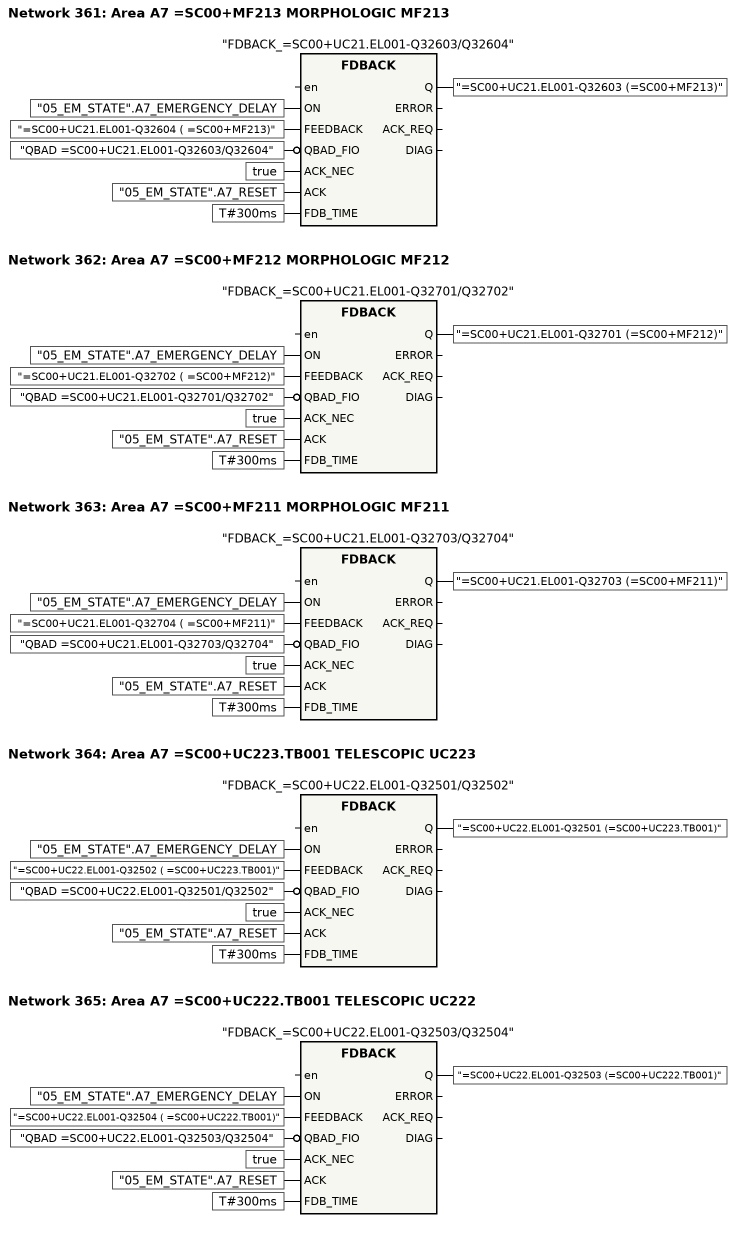
   "FDBACK_=SC00+UC21.EL001-Q32603/Q32604"(ON := "05_EM_STATE".A7_EMERGENCY_DELAY,   // FDBACK
                           FEEDBACK := "=SC00+UC21.EL001-Q32604 ( =SC00+MF213)",
                           QBAD_FIO := NOT "QBAD =SC00+UC21.EL001-Q32603/Q32604",
                           ACK_NEC := true,
                           ACK := "05_EM_STATE".A7_RESET,
                           FDB_TIME := T#300ms,
                           Q => "=SC00+UC21.EL001-Q32603 (=SC00+MF213)");
END_REGION

REGION Network 362: Area A7 =SC00+MF212 MORPHOLOGIC MF212
   "FDBACK_=SC00+UC21.EL001-Q32701/Q32702"(ON := "05_EM_STATE".A7_EMERGENCY_DELAY,   // FDBACK
                           FEEDBACK := "=SC00+UC21.EL001-Q32702 ( =SC00+MF212)",
                           QBAD_FIO := NOT "QBAD =SC00+UC21.EL001-Q32701/Q32702",
                           ACK_NEC := true,
                           ACK := "05_EM_STATE".A7_RESET,
                           FDB_TIME := T#300ms,
                           Q => "=SC00+UC21.EL001-Q32701 (=SC00+MF212)");
END_REGION

REGION Network 363: Area A7 =SC00+MF211 MORPHOLOGIC MF211
   "FDBACK_=SC00+UC21.EL001-Q32703/Q32704"(ON := "05_EM_STATE".A7_EMERGENCY_DELAY,   // FDBACK
                           FEEDBACK := "=SC00+UC21.EL001-Q32704 ( =SC00+MF211)",
                           QBAD_FIO := NOT "QBAD =SC00+UC21.EL001-Q32703/Q32704",
                           ACK_NEC := true,
                           ACK := "05_EM_STATE".A7_RESET,
                           FDB_TIME := T#300ms,
                           Q => "=SC00+UC21.EL001-Q32703 (=SC00+MF211)");
END_REGION

REGION Network 364: Area A7 =SC00+UC223.TB001 TELESCOPIC UC223
   "FDBACK_=SC00+UC22.EL001-Q32501/Q32502"(ON := "05_EM_STATE".A7_EMERGENCY_DELAY,   // FDBACK
                           FEEDBACK := "=SC00+UC22.EL001-Q32502 ( =SC00+UC223.TB001)",
                           QBAD_FIO := NOT "QBAD =SC00+UC22.EL001-Q32501/Q32502",
                           ACK_NEC := true,
                           ACK := "05_EM_STATE".A7_RESET,
                           FDB_TIME := T#300ms,
                           Q => "=SC00+UC22.EL001-Q32501 (=SC00+UC223.TB001)");
END_REGION

REGION Network 365: Area A7 =SC00+UC222.TB001 TELESCOPIC UC222
   "FDBACK_=SC00+UC22.EL001-Q32503/Q32504"(ON := "05_EM_STATE".A7_EMERGENCY_DELAY,   // FDBACK
                           FEEDBACK := "=SC00+UC22.EL001-Q32504 ( =SC00+UC222.TB001)",
                           QBAD_FIO := NOT "QBAD =SC00+UC22.EL001-Q32503/Q32504",
                           ACK_NEC := true,
                           ACK := "05_EM_STATE".A7_RESET,
                           FDB_TIME := T#300ms,
                           Q => "=SC00+UC22.EL001-Q32503 (=SC00+UC222.TB001)");
END_REGION

REGION Network 366: Area A7 =SC00+UC221.TB001 TELESCOPIC UC221
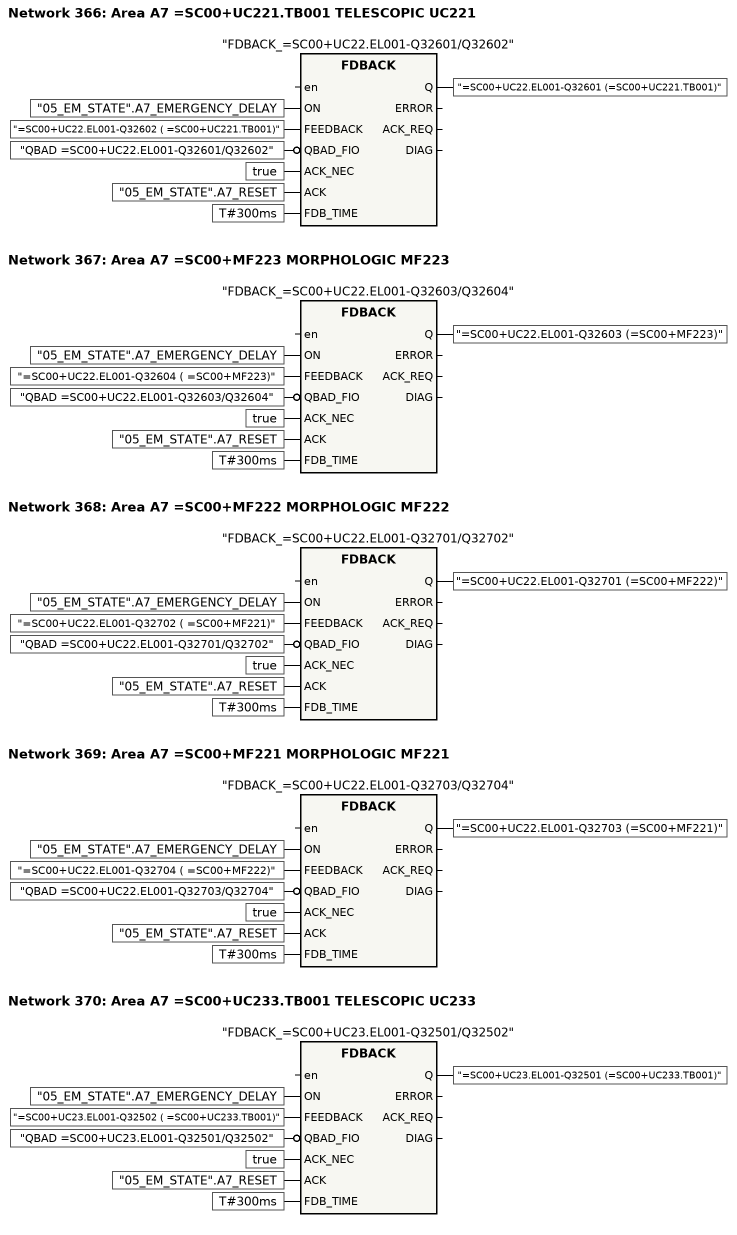
   "FDBACK_=SC00+UC22.EL001-Q32601/Q32602"(ON := "05_EM_STATE".A7_EMERGENCY_DELAY,   // FDBACK
                           FEEDBACK := "=SC00+UC22.EL001-Q32602 ( =SC00+UC221.TB001)",
                           QBAD_FIO := NOT "QBAD =SC00+UC22.EL001-Q32601/Q32602",
                           ACK_NEC := true,
                           ACK := "05_EM_STATE".A7_RESET,
                           FDB_TIME := T#300ms,
                           Q => "=SC00+UC22.EL001-Q32601 (=SC00+UC221.TB001)");
END_REGION

REGION Network 367: Area A7 =SC00+MF223 MORPHOLOGIC MF223
   "FDBACK_=SC00+UC22.EL001-Q32603/Q32604"(ON := "05_EM_STATE".A7_EMERGENCY_DELAY,   // FDBACK
                           FEEDBACK := "=SC00+UC22.EL001-Q32604 ( =SC00+MF223)",
                           QBAD_FIO := NOT "QBAD =SC00+UC22.EL001-Q32603/Q32604",
                           ACK_NEC := true,
                           ACK := "05_EM_STATE".A7_RESET,
                           FDB_TIME := T#300ms,
                           Q => "=SC00+UC22.EL001-Q32603 (=SC00+MF223)");
END_REGION

REGION Network 368: Area A7 =SC00+MF222 MORPHOLOGIC MF222
   "FDBACK_=SC00+UC22.EL001-Q32701/Q32702"(ON := "05_EM_STATE".A7_EMERGENCY_DELAY,   // FDBACK
                           FEEDBACK := "=SC00+UC22.EL001-Q32702 ( =SC00+MF221)",
                           QBAD_FIO := NOT "QBAD =SC00+UC22.EL001-Q32701/Q32702",
                           ACK_NEC := true,
                           ACK := "05_EM_STATE".A7_RESET,
                           FDB_TIME := T#300ms,
                           Q => "=SC00+UC22.EL001-Q32701 (=SC00+MF222)");
END_REGION

REGION Network 369: Area A7 =SC00+MF221 MORPHOLOGIC MF221
   "FDBACK_=SC00+UC22.EL001-Q32703/Q32704"(ON := "05_EM_STATE".A7_EMERGENCY_DELAY,   // FDBACK
                           FEEDBACK := "=SC00+UC22.EL001-Q32704 ( =SC00+MF222)",
                           QBAD_FIO := NOT "QBAD =SC00+UC22.EL001-Q32703/Q32704",
                           ACK_NEC := true,
                           ACK := "05_EM_STATE".A7_RESET,
                           FDB_TIME := T#300ms,
                           Q => "=SC00+UC22.EL001-Q32703 (=SC00+MF221)");
END_REGION

REGION Network 370: Area A7 =SC00+UC233.TB001 TELESCOPIC UC233
   "FDBACK_=SC00+UC23.EL001-Q32501/Q32502"(ON := "05_EM_STATE".A7_EMERGENCY_DELAY,   // FDBACK
                           FEEDBACK := "=SC00+UC23.EL001-Q32502 ( =SC00+UC233.TB001)",
                           QBAD_FIO := NOT "QBAD =SC00+UC23.EL001-Q32501/Q32502",
                           ACK_NEC := true,
                           ACK := "05_EM_STATE".A7_RESET,
                           FDB_TIME := T#300ms,
                           Q => "=SC00+UC23.EL001-Q32501 (=SC00+UC233.TB001)");
END_REGION

REGION Network 371: Area A7 =SC00+UC232.TB001 TELESCOPIC UC232
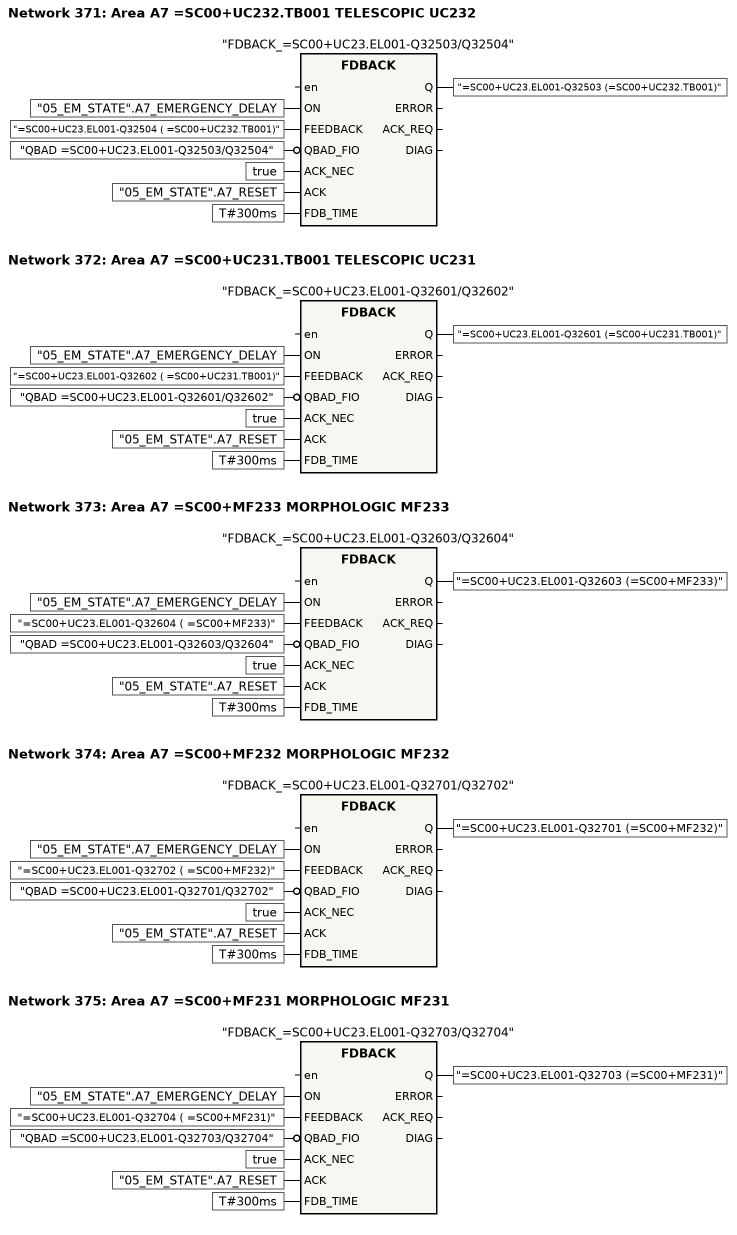
   "FDBACK_=SC00+UC23.EL001-Q32503/Q32504"(ON := "05_EM_STATE".A7_EMERGENCY_DELAY,   // FDBACK
                           FEEDBACK := "=SC00+UC23.EL001-Q32504 ( =SC00+UC232.TB001)",
                           QBAD_FIO := NOT "QBAD =SC00+UC23.EL001-Q32503/Q32504",
                           ACK_NEC := true,
                           ACK := "05_EM_STATE".A7_RESET,
                           FDB_TIME := T#300ms,
                           Q => "=SC00+UC23.EL001-Q32503 (=SC00+UC232.TB001)");
END_REGION

REGION Network 372: Area A7 =SC00+UC231.TB001 TELESCOPIC UC231
   "FDBACK_=SC00+UC23.EL001-Q32601/Q32602"(ON := "05_EM_STATE".A7_EMERGENCY_DELAY,   // FDBACK
                           FEEDBACK := "=SC00+UC23.EL001-Q32602 ( =SC00+UC231.TB001)",
                           QBAD_FIO := NOT "QBAD =SC00+UC23.EL001-Q32601/Q32602",
                           ACK_NEC := true,
                           ACK := "05_EM_STATE".A7_RESET,
                           FDB_TIME := T#300ms,
                           Q => "=SC00+UC23.EL001-Q32601 (=SC00+UC231.TB001)");
END_REGION

REGION Network 373: Area A7 =SC00+MF233 MORPHOLOGIC MF233
   "FDBACK_=SC00+UC23.EL001-Q32603/Q32604"(ON := "05_EM_STATE".A7_EMERGENCY_DELAY,   // FDBACK
                           FEEDBACK := "=SC00+UC23.EL001-Q32604 ( =SC00+MF233)",
                           QBAD_FIO := NOT "QBAD =SC00+UC23.EL001-Q32603/Q32604",
                           ACK_NEC := true,
                           ACK := "05_EM_STATE".A7_RESET,
                           FDB_TIME := T#300ms,
                           Q => "=SC00+UC23.EL001-Q32603 (=SC00+MF233)");
END_REGION

REGION Network 374: Area A7 =SC00+MF232 MORPHOLOGIC MF232
   "FDBACK_=SC00+UC23.EL001-Q32701/Q32702"(ON := "05_EM_STATE".A7_EMERGENCY_DELAY,   // FDBACK
                           FEEDBACK := "=SC00+UC23.EL001-Q32702 ( =SC00+MF232)",
                           QBAD_FIO := NOT "QBAD =SC00+UC23.EL001-Q32701/Q32702",
                           ACK_NEC := true,
                           ACK := "05_EM_STATE".A7_RESET,
                           FDB_TIME := T#300ms,
                           Q => "=SC00+UC23.EL001-Q32701 (=SC00+MF232)");
END_REGION

REGION Network 375: Area A7 =SC00+MF231 MORPHOLOGIC MF231
   "FDBACK_=SC00+UC23.EL001-Q32703/Q32704"(ON := "05_EM_STATE".A7_EMERGENCY_DELAY,   // FDBACK
                           FEEDBACK := "=SC00+UC23.EL001-Q32704 ( =SC00+MF231)",
                           QBAD_FIO := NOT "QBAD =SC00+UC23.EL001-Q32703/Q32704",
                           ACK_NEC := true,
                           ACK := "05_EM_STATE".A7_RESET,
                           FDB_TIME := T#300ms,
                           Q => "=SC00+UC23.EL001-Q32703 (=SC00+MF231)");
END_REGION

REGION Network 376: Area A7 =SC00+UC243.TB001 TELESCOPIC UC243
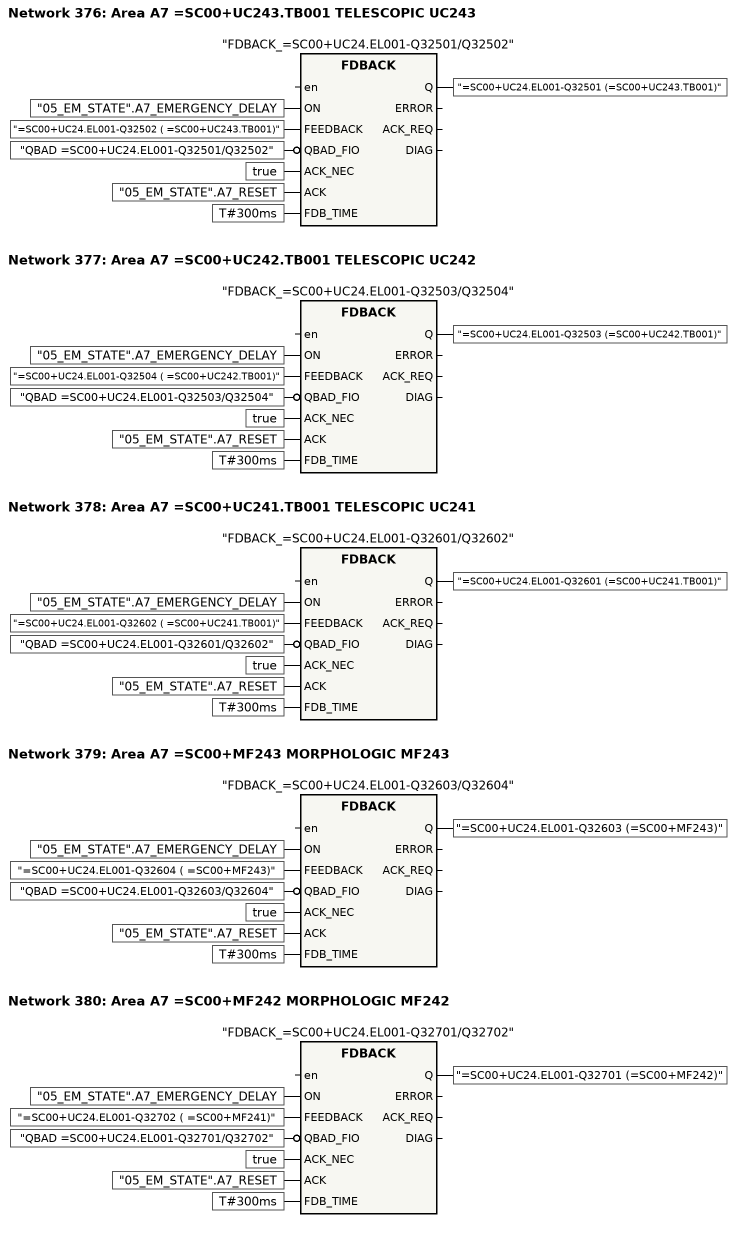
   "FDBACK_=SC00+UC24.EL001-Q32501/Q32502"(ON := "05_EM_STATE".A7_EMERGENCY_DELAY,   // FDBACK
                           FEEDBACK := "=SC00+UC24.EL001-Q32502 ( =SC00+UC243.TB001)",
                           QBAD_FIO := NOT "QBAD =SC00+UC24.EL001-Q32501/Q32502",
                           ACK_NEC := true,
                           ACK := "05_EM_STATE".A7_RESET,
                           FDB_TIME := T#300ms,
                           Q => "=SC00+UC24.EL001-Q32501 (=SC00+UC243.TB001)");
END_REGION

REGION Network 377: Area A7 =SC00+UC242.TB001 TELESCOPIC UC242
   "FDBACK_=SC00+UC24.EL001-Q32503/Q32504"(ON := "05_EM_STATE".A7_EMERGENCY_DELAY,   // FDBACK
                           FEEDBACK := "=SC00+UC24.EL001-Q32504 ( =SC00+UC242.TB001)",
                           QBAD_FIO := NOT "QBAD =SC00+UC24.EL001-Q32503/Q32504",
                           ACK_NEC := true,
                           ACK := "05_EM_STATE".A7_RESET,
                           FDB_TIME := T#300ms,
                           Q => "=SC00+UC24.EL001-Q32503 (=SC00+UC242.TB001)");
END_REGION

REGION Network 378: Area A7 =SC00+UC241.TB001 TELESCOPIC UC241
   "FDBACK_=SC00+UC24.EL001-Q32601/Q32602"(ON := "05_EM_STATE".A7_EMERGENCY_DELAY,   // FDBACK
                           FEEDBACK := "=SC00+UC24.EL001-Q32602 ( =SC00+UC241.TB001)",
                           QBAD_FIO := NOT "QBAD =SC00+UC24.EL001-Q32601/Q32602",
                           ACK_NEC := true,
                           ACK := "05_EM_STATE".A7_RESET,
                           FDB_TIME := T#300ms,
                           Q => "=SC00+UC24.EL001-Q32601 (=SC00+UC241.TB001)");
END_REGION

REGION Network 379: Area A7 =SC00+MF243 MORPHOLOGIC MF243
   "FDBACK_=SC00+UC24.EL001-Q32603/Q32604"(ON := "05_EM_STATE".A7_EMERGENCY_DELAY,   // FDBACK
                           FEEDBACK := "=SC00+UC24.EL001-Q32604 ( =SC00+MF243)",
                           QBAD_FIO := NOT "QBAD =SC00+UC24.EL001-Q32603/Q32604",
                           ACK_NEC := true,
                           ACK := "05_EM_STATE".A7_RESET,
                           FDB_TIME := T#300ms,
                           Q => "=SC00+UC24.EL001-Q32603 (=SC00+MF243)");
END_REGION

REGION Network 380: Area A7 =SC00+MF242 MORPHOLOGIC MF242
   "FDBACK_=SC00+UC24.EL001-Q32701/Q32702"(ON := "05_EM_STATE".A7_EMERGENCY_DELAY,   // FDBACK
                           FEEDBACK := "=SC00+UC24.EL001-Q32702 ( =SC00+MF241)",
                           QBAD_FIO := NOT "QBAD =SC00+UC24.EL001-Q32701/Q32702",
                           ACK_NEC := true,
                           ACK := "05_EM_STATE".A7_RESET,
                           FDB_TIME := T#300ms,
                           Q => "=SC00+UC24.EL001-Q32701 (=SC00+MF242)");
END_REGION

REGION Network 381: Area A7 =SC00+MF241 MORPHOLOGIC MF241
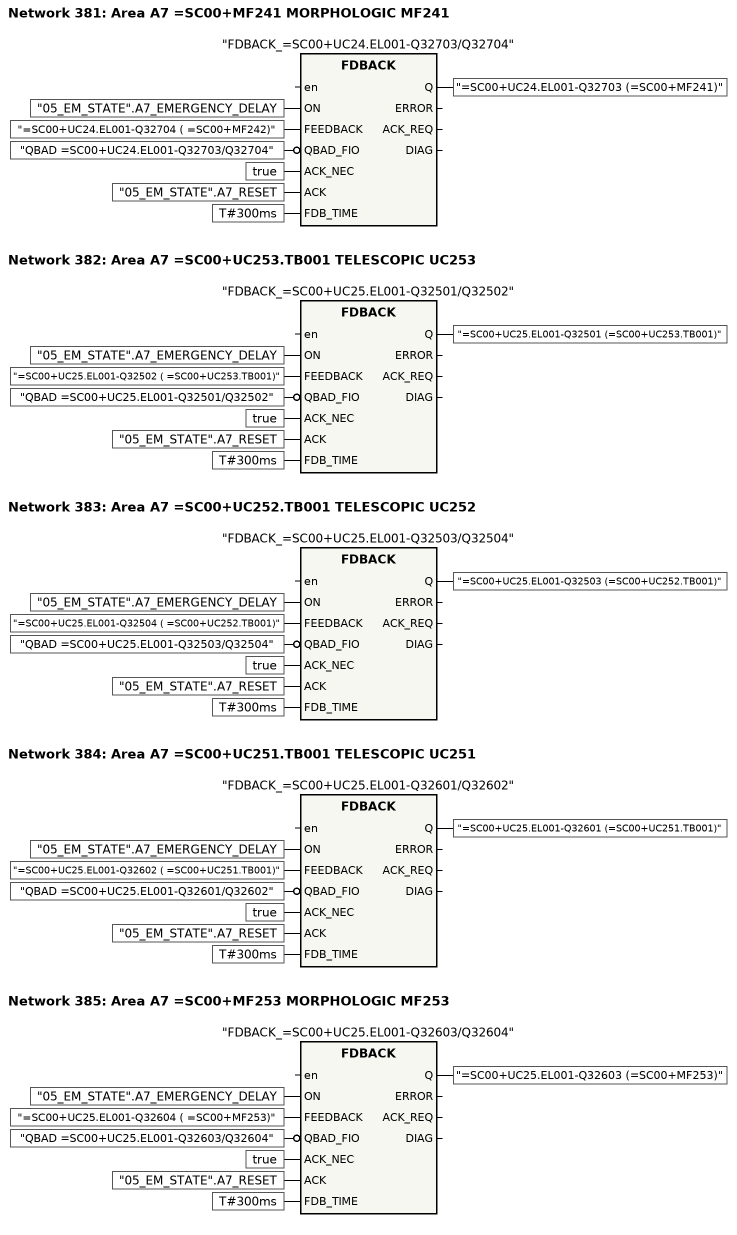
   "FDBACK_=SC00+UC24.EL001-Q32703/Q32704"(ON := "05_EM_STATE".A7_EMERGENCY_DELAY,   // FDBACK
                           FEEDBACK := "=SC00+UC24.EL001-Q32704 ( =SC00+MF242)",
                           QBAD_FIO := NOT "QBAD =SC00+UC24.EL001-Q32703/Q32704",
                           ACK_NEC := true,
                           ACK := "05_EM_STATE".A7_RESET,
                           FDB_TIME := T#300ms,
                           Q => "=SC00+UC24.EL001-Q32703 (=SC00+MF241)");
END_REGION

REGION Network 382: Area A7 =SC00+UC253.TB001 TELESCOPIC UC253
   "FDBACK_=SC00+UC25.EL001-Q32501/Q32502"(ON := "05_EM_STATE".A7_EMERGENCY_DELAY,   // FDBACK
                           FEEDBACK := "=SC00+UC25.EL001-Q32502 ( =SC00+UC253.TB001)",
                           QBAD_FIO := NOT "QBAD =SC00+UC25.EL001-Q32501/Q32502",
                           ACK_NEC := true,
                           ACK := "05_EM_STATE".A7_RESET,
                           FDB_TIME := T#300ms,
                           Q => "=SC00+UC25.EL001-Q32501 (=SC00+UC253.TB001)");
END_REGION

REGION Network 383: Area A7 =SC00+UC252.TB001 TELESCOPIC UC252
   "FDBACK_=SC00+UC25.EL001-Q32503/Q32504"(ON := "05_EM_STATE".A7_EMERGENCY_DELAY,   // FDBACK
                           FEEDBACK := "=SC00+UC25.EL001-Q32504 ( =SC00+UC252.TB001)",
                           QBAD_FIO := NOT "QBAD =SC00+UC25.EL001-Q32503/Q32504",
                           ACK_NEC := true,
                           ACK := "05_EM_STATE".A7_RESET,
                           FDB_TIME := T#300ms,
                           Q => "=SC00+UC25.EL001-Q32503 (=SC00+UC252.TB001)");
END_REGION

REGION Network 384: Area A7 =SC00+UC251.TB001 TELESCOPIC UC251
   "FDBACK_=SC00+UC25.EL001-Q32601/Q32602"(ON := "05_EM_STATE".A7_EMERGENCY_DELAY,   // FDBACK
                           FEEDBACK := "=SC00+UC25.EL001-Q32602 ( =SC00+UC251.TB001)",
                           QBAD_FIO := NOT "QBAD =SC00+UC25.EL001-Q32601/Q32602",
                           ACK_NEC := true,
                           ACK := "05_EM_STATE".A7_RESET,
                           FDB_TIME := T#300ms,
                           Q => "=SC00+UC25.EL001-Q32601 (=SC00+UC251.TB001)");
END_REGION

REGION Network 385: Area A7 =SC00+MF253 MORPHOLOGIC MF253
   "FDBACK_=SC00+UC25.EL001-Q32603/Q32604"(ON := "05_EM_STATE".A7_EMERGENCY_DELAY,   // FDBACK
                           FEEDBACK := "=SC00+UC25.EL001-Q32604 ( =SC00+MF253)",
                           QBAD_FIO := NOT "QBAD =SC00+UC25.EL001-Q32603/Q32604",
                           ACK_NEC := true,
                           ACK := "05_EM_STATE".A7_RESET,
                           FDB_TIME := T#300ms,
                           Q => "=SC00+UC25.EL001-Q32603 (=SC00+MF253)");
END_REGION

REGION Network 386: Area A7 =SC00+MF252 MORPHOLOGIC MF252
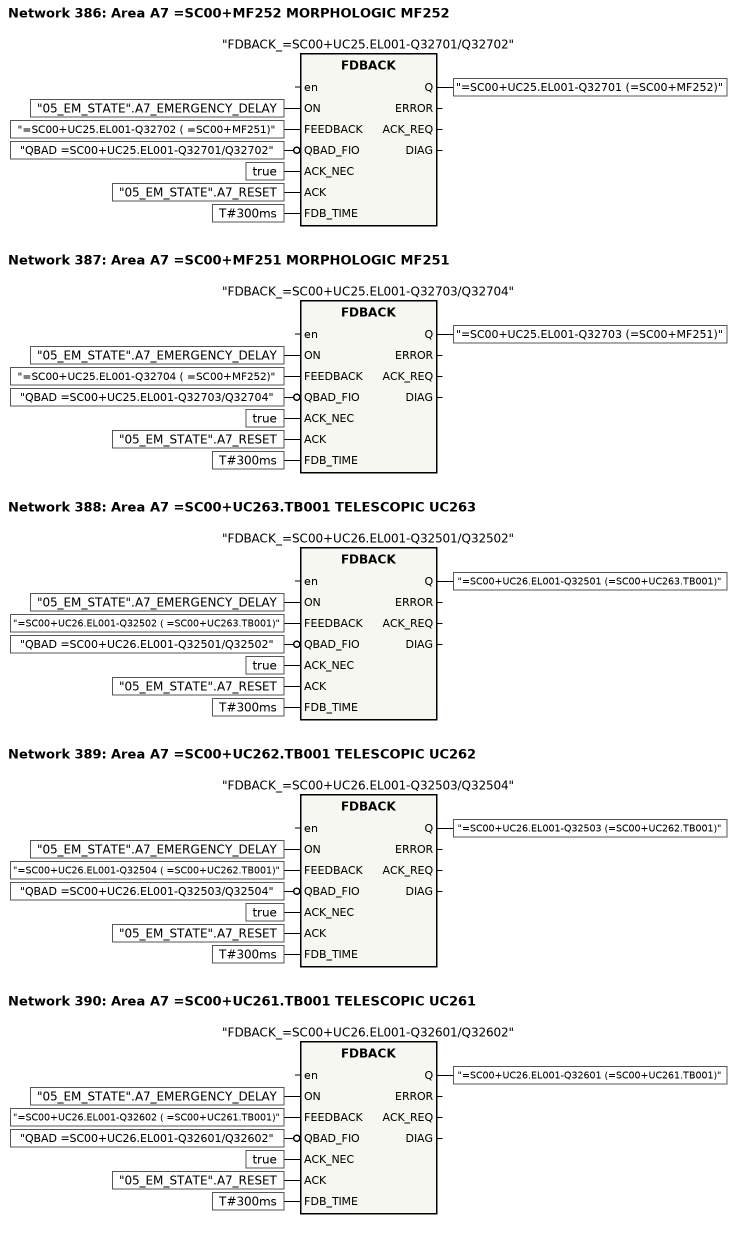
   "FDBACK_=SC00+UC25.EL001-Q32701/Q32702"(ON := "05_EM_STATE".A7_EMERGENCY_DELAY,   // FDBACK
                           FEEDBACK := "=SC00+UC25.EL001-Q32702 ( =SC00+MF251)",
                           QBAD_FIO := NOT "QBAD =SC00+UC25.EL001-Q32701/Q32702",
                           ACK_NEC := true,
                           ACK := "05_EM_STATE".A7_RESET,
                           FDB_TIME := T#300ms,
                           Q => "=SC00+UC25.EL001-Q32701 (=SC00+MF252)");
END_REGION

REGION Network 387: Area A7 =SC00+MF251 MORPHOLOGIC MF251
   "FDBACK_=SC00+UC25.EL001-Q32703/Q32704"(ON := "05_EM_STATE".A7_EMERGENCY_DELAY,   // FDBACK
                           FEEDBACK := "=SC00+UC25.EL001-Q32704 ( =SC00+MF252)",
                           QBAD_FIO := NOT "QBAD =SC00+UC25.EL001-Q32703/Q32704",
                           ACK_NEC := true,
                           ACK := "05_EM_STATE".A7_RESET,
                           FDB_TIME := T#300ms,
                           Q => "=SC00+UC25.EL001-Q32703 (=SC00+MF251)");
END_REGION

REGION Network 388: Area A7 =SC00+UC263.TB001 TELESCOPIC UC263
   "FDBACK_=SC00+UC26.EL001-Q32501/Q32502"(ON := "05_EM_STATE".A7_EMERGENCY_DELAY,   // FDBACK
                           FEEDBACK := "=SC00+UC26.EL001-Q32502 ( =SC00+UC263.TB001)",
                           QBAD_FIO := NOT "QBAD =SC00+UC26.EL001-Q32501/Q32502",
                           ACK_NEC := true,
                           ACK := "05_EM_STATE".A7_RESET,
                           FDB_TIME := T#300ms,
                           Q => "=SC00+UC26.EL001-Q32501 (=SC00+UC263.TB001)");
END_REGION

REGION Network 389: Area A7 =SC00+UC262.TB001 TELESCOPIC UC262
   "FDBACK_=SC00+UC26.EL001-Q32503/Q32504"(ON := "05_EM_STATE".A7_EMERGENCY_DELAY,   // FDBACK
                           FEEDBACK := "=SC00+UC26.EL001-Q32504 ( =SC00+UC262.TB001)",
                           QBAD_FIO := NOT "QBAD =SC00+UC26.EL001-Q32503/Q32504",
                           ACK_NEC := true,
                           ACK := "05_EM_STATE".A7_RESET,
                           FDB_TIME := T#300ms,
                           Q => "=SC00+UC26.EL001-Q32503 (=SC00+UC262.TB001)");
END_REGION

REGION Network 390: Area A7 =SC00+UC261.TB001 TELESCOPIC UC261
   "FDBACK_=SC00+UC26.EL001-Q32601/Q32602"(ON := "05_EM_STATE".A7_EMERGENCY_DELAY,   // FDBACK
                           FEEDBACK := "=SC00+UC26.EL001-Q32602 ( =SC00+UC261.TB001)",
                           QBAD_FIO := NOT "QBAD =SC00+UC26.EL001-Q32601/Q32602",
                           ACK_NEC := true,
                           ACK := "05_EM_STATE".A7_RESET,
                           FDB_TIME := T#300ms,
                           Q => "=SC00+UC26.EL001-Q32601 (=SC00+UC261.TB001)");
END_REGION

REGION Network 391: Area A7 =SC00+MF263 MORPHOLOGIC MF263
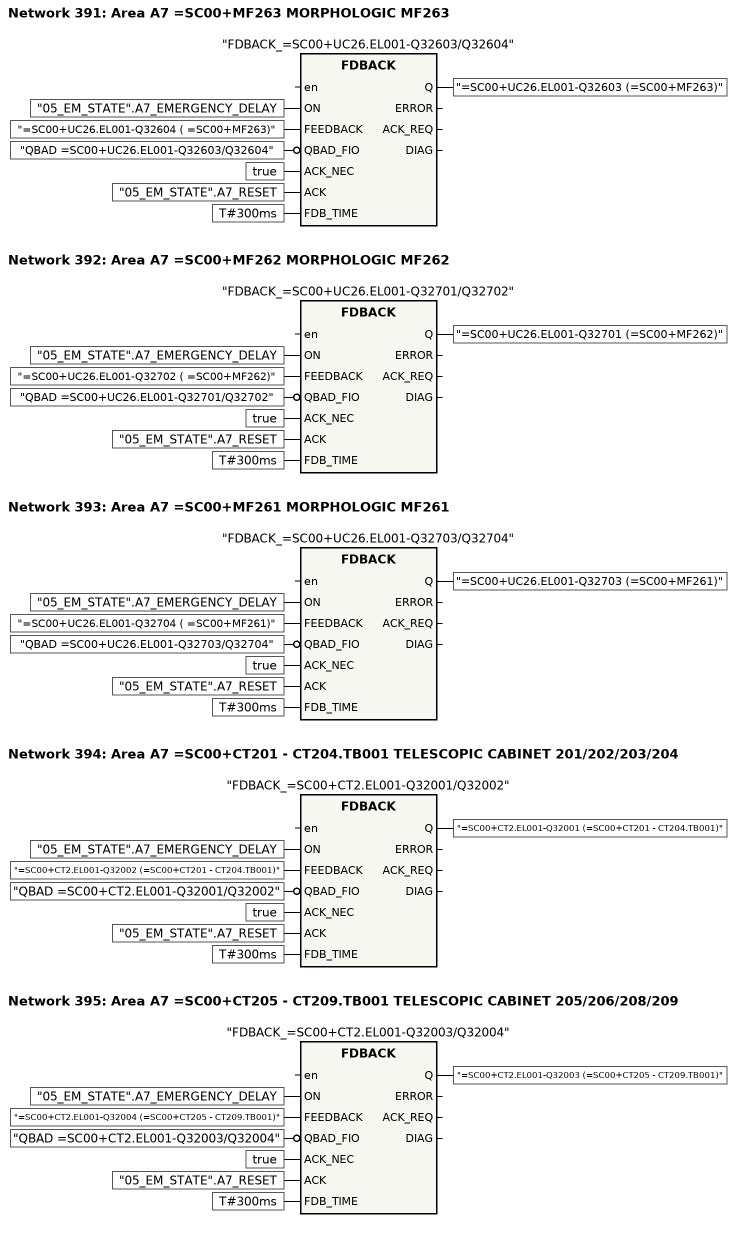
   "FDBACK_=SC00+UC26.EL001-Q32603/Q32604"(ON := "05_EM_STATE".A7_EMERGENCY_DELAY,   // FDBACK
                           FEEDBACK := "=SC00+UC26.EL001-Q32604 ( =SC00+MF263)",
                           QBAD_FIO := NOT "QBAD =SC00+UC26.EL001-Q32603/Q32604",
                           ACK_NEC := true,
                           ACK := "05_EM_STATE".A7_RESET,
                           FDB_TIME := T#300ms,
                           Q => "=SC00+UC26.EL001-Q32603 (=SC00+MF263)");
END_REGION

REGION Network 392: Area A7 =SC00+MF262 MORPHOLOGIC MF262
   "FDBACK_=SC00+UC26.EL001-Q32701/Q32702"(ON := "05_EM_STATE".A7_EMERGENCY_DELAY,   // FDBACK
                           FEEDBACK := "=SC00+UC26.EL001-Q32702 ( =SC00+MF262)",
                           QBAD_FIO := NOT "QBAD =SC00+UC26.EL001-Q32701/Q32702",
                           ACK_NEC := true,
                           ACK := "05_EM_STATE".A7_RESET,
                           FDB_TIME := T#300ms,
                           Q => "=SC00+UC26.EL001-Q32701 (=SC00+MF262)");
END_REGION

REGION Network 393: Area A7 =SC00+MF261 MORPHOLOGIC MF261
   "FDBACK_=SC00+UC26.EL001-Q32703/Q32704"(ON := "05_EM_STATE".A7_EMERGENCY_DELAY,   // FDBACK
                           FEEDBACK := "=SC00+UC26.EL001-Q32704 ( =SC00+MF261)",
                           QBAD_FIO := NOT "QBAD =SC00+UC26.EL001-Q32703/Q32704",
                           ACK_NEC := true,
                           ACK := "05_EM_STATE".A7_RESET,
                           FDB_TIME := T#300ms,
                           Q => "=SC00+UC26.EL001-Q32703 (=SC00+MF261)");
END_REGION

REGION Network 394: Area A7 =SC00+CT201 - CT204.TB001 TELESCOPIC CABINET 201/202/203/204
   "FDBACK_=SC00+CT2.EL001-Q32001/Q32002"(ON := "05_EM_STATE".A7_EMERGENCY_DELAY,   // FDBACK
                           FEEDBACK := "=SC00+CT2.EL001-Q32002 (=SC00+CT201 - CT204.TB001)",
                           QBAD_FIO := NOT "QBAD =SC00+CT2.EL001-Q32001/Q32002",
                           ACK_NEC := true,
                           ACK := "05_EM_STATE".A7_RESET,
                           FDB_TIME := T#300ms,
                           Q => "=SC00+CT2.EL001-Q32001 (=SC00+CT201 - CT204.TB001)");
END_REGION

REGION Network 395: Area A7 =SC00+CT205 - CT209.TB001 TELESCOPIC CABINET 205/206/208/209
   "FDBACK_=SC00+CT2.EL001-Q32003/Q32004"(ON := "05_EM_STATE".A7_EMERGENCY_DELAY,   // FDBACK
                           FEEDBACK := "=SC00+CT2.EL001-Q32004 (=SC00+CT205 - CT209.TB001)",
                           QBAD_FIO := NOT "QBAD =SC00+CT2.EL001-Q32003/Q32004",
                           ACK_NEC := true,
                           ACK := "05_EM_STATE".A7_RESET,
                           FDB_TIME := T#300ms,
                           Q => "=SC00+CT2.EL001-Q32003 (=SC00+CT205 - CT209.TB001)");
END_REGION

REGION Network 396: Area A7 =SC00+CT210 - CT213.TB001 TELESCOPIC CABINET 210/211/212/213
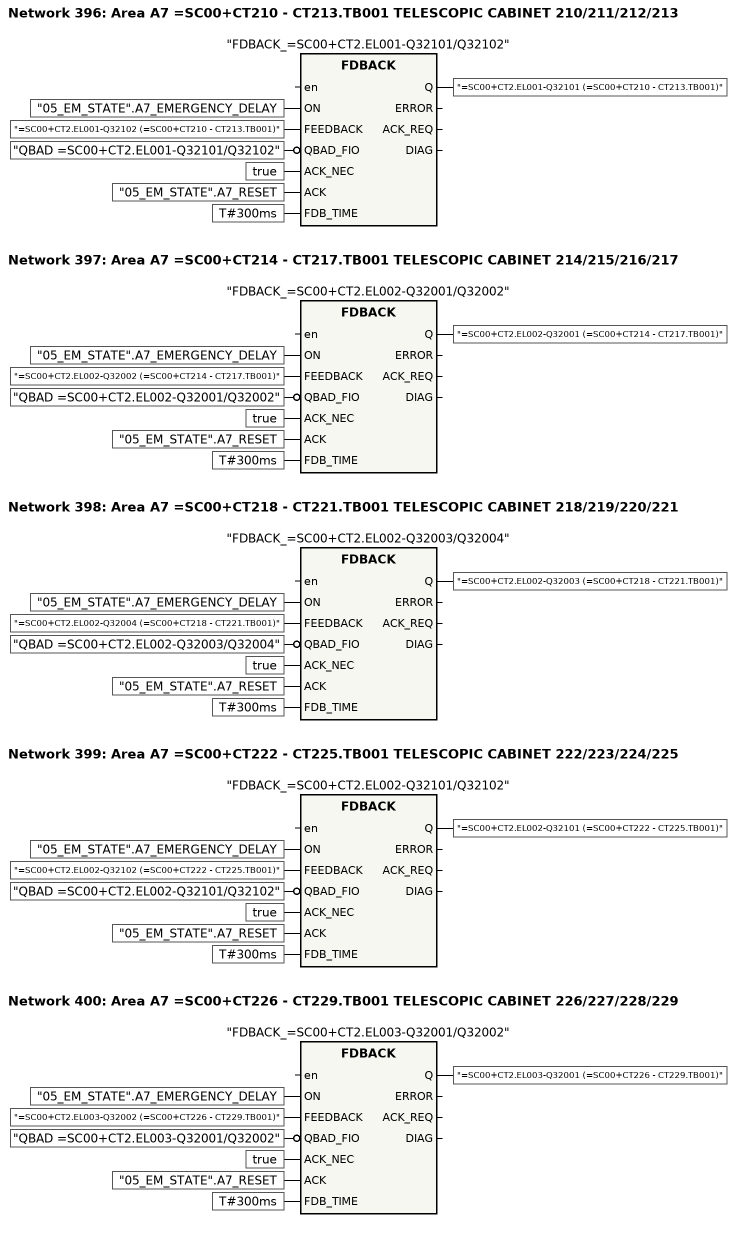
   "FDBACK_=SC00+CT2.EL001-Q32101/Q32102"(ON := "05_EM_STATE".A7_EMERGENCY_DELAY,   // FDBACK
                           FEEDBACK := "=SC00+CT2.EL001-Q32102 (=SC00+CT210 - CT213.TB001)",
                           QBAD_FIO := NOT "QBAD =SC00+CT2.EL001-Q32101/Q32102",
                           ACK_NEC := true,
                           ACK := "05_EM_STATE".A7_RESET,
                           FDB_TIME := T#300ms,
                           Q => "=SC00+CT2.EL001-Q32101 (=SC00+CT210 - CT213.TB001)");
END_REGION

REGION Network 397: Area A7 =SC00+CT214 - CT217.TB001 TELESCOPIC CABINET 214/215/216/217
   "FDBACK_=SC00+CT2.EL002-Q32001/Q32002"(ON := "05_EM_STATE".A7_EMERGENCY_DELAY,   // FDBACK
                           FEEDBACK := "=SC00+CT2.EL002-Q32002 (=SC00+CT214 - CT217.TB001)",
                           QBAD_FIO := NOT "QBAD =SC00+CT2.EL002-Q32001/Q32002",
                           ACK_NEC := true,
                           ACK := "05_EM_STATE".A7_RESET,
                           FDB_TIME := T#300ms,
                           Q => "=SC00+CT2.EL002-Q32001 (=SC00+CT214 - CT217.TB001)");
END_REGION

REGION Network 398: Area A7 =SC00+CT218 - CT221.TB001 TELESCOPIC CABINET 218/219/220/221
   "FDBACK_=SC00+CT2.EL002-Q32003/Q32004"(ON := "05_EM_STATE".A7_EMERGENCY_DELAY,   // FDBACK
                           FEEDBACK := "=SC00+CT2.EL002-Q32004 (=SC00+CT218 - CT221.TB001)",
                           QBAD_FIO := NOT "QBAD =SC00+CT2.EL002-Q32003/Q32004",
                           ACK_NEC := true,
                           ACK := "05_EM_STATE".A7_RESET,
                           FDB_TIME := T#300ms,
                           Q => "=SC00+CT2.EL002-Q32003 (=SC00+CT218 - CT221.TB001)");
END_REGION

REGION Network 399: Area A7 =SC00+CT222 - CT225.TB001 TELESCOPIC CABINET 222/223/224/225
   "FDBACK_=SC00+CT2.EL002-Q32101/Q32102"(ON := "05_EM_STATE".A7_EMERGENCY_DELAY,   // FDBACK
                           FEEDBACK := "=SC00+CT2.EL002-Q32102 (=SC00+CT222 - CT225.TB001)",
                           QBAD_FIO := NOT "QBAD =SC00+CT2.EL002-Q32101/Q32102",
                           ACK_NEC := true,
                           ACK := "05_EM_STATE".A7_RESET,
                           FDB_TIME := T#300ms,
                           Q => "=SC00+CT2.EL002-Q32101 (=SC00+CT222 - CT225.TB001)");
END_REGION

REGION Network 400: Area A7 =SC00+CT226 - CT229.TB001 TELESCOPIC CABINET 226/227/228/229
   "FDBACK_=SC00+CT2.EL003-Q32001/Q32002"(ON := "05_EM_STATE".A7_EMERGENCY_DELAY,   // FDBACK
                           FEEDBACK := "=SC00+CT2.EL003-Q32002 (=SC00+CT226 - CT229.TB001)",
                           QBAD_FIO := NOT "QBAD =SC00+CT2.EL003-Q32001/Q32002",
                           ACK_NEC := true,
                           ACK := "05_EM_STATE".A7_RESET,
                           FDB_TIME := T#300ms,
                           Q => "=SC00+CT2.EL003-Q32001 (=SC00+CT226 - CT229.TB001)");
END_REGION

REGION Network 401: Area A7 =SC00+CT230 - CT233.TB001 TELESCOPIC CABINET 230/231/232/233
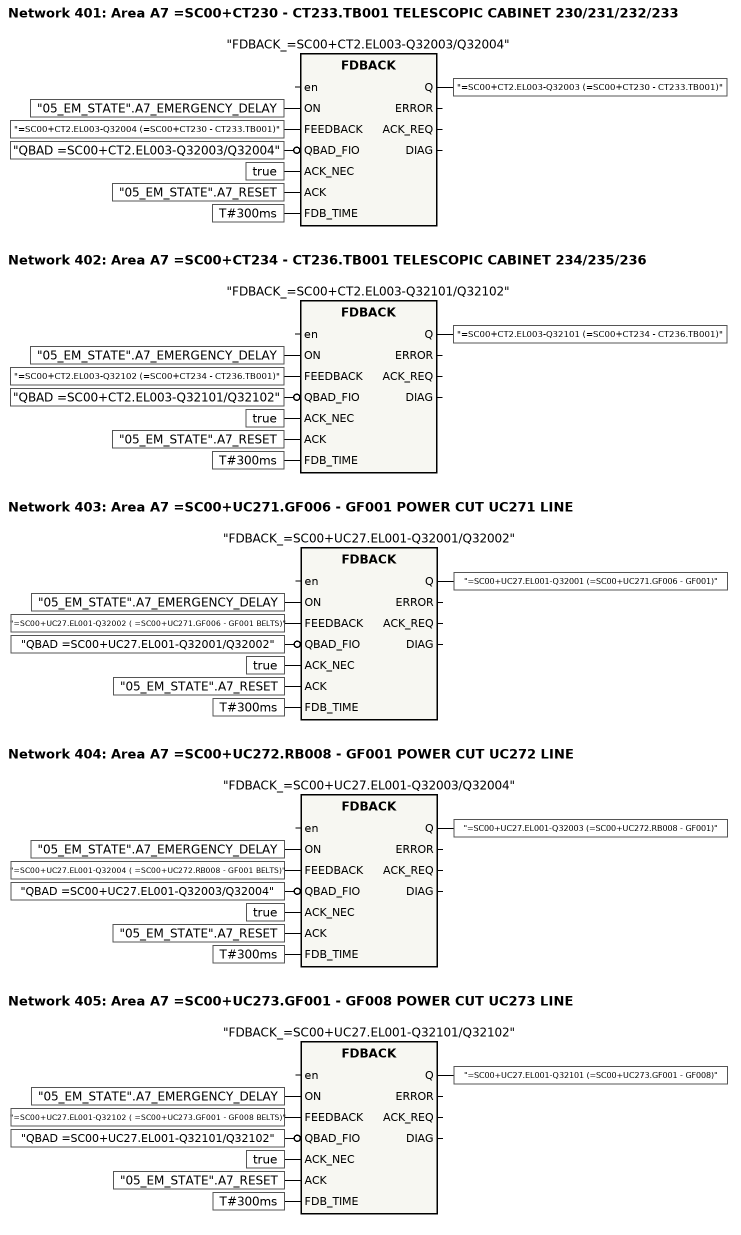
   "FDBACK_=SC00+CT2.EL003-Q32003/Q32004"(ON := "05_EM_STATE".A7_EMERGENCY_DELAY,   // FDBACK
                           FEEDBACK := "=SC00+CT2.EL003-Q32004 (=SC00+CT230 - CT233.TB001)",
                           QBAD_FIO := NOT "QBAD =SC00+CT2.EL003-Q32003/Q32004",
                           ACK_NEC := true,
                           ACK := "05_EM_STATE".A7_RESET,
                           FDB_TIME := T#300ms,
                           Q => "=SC00+CT2.EL003-Q32003 (=SC00+CT230 - CT233.TB001)");
END_REGION

REGION Network 402: Area A7 =SC00+CT234 - CT236.TB001 TELESCOPIC CABINET 234/235/236
   "FDBACK_=SC00+CT2.EL003-Q32101/Q32102"(ON := "05_EM_STATE".A7_EMERGENCY_DELAY,   // FDBACK
                           FEEDBACK := "=SC00+CT2.EL003-Q32102 (=SC00+CT234 - CT236.TB001)",
                           QBAD_FIO := NOT "QBAD =SC00+CT2.EL003-Q32101/Q32102",
                           ACK_NEC := true,
                           ACK := "05_EM_STATE".A7_RESET,
                           FDB_TIME := T#300ms,
                           Q => "=SC00+CT2.EL003-Q32101 (=SC00+CT234 - CT236.TB001)");
END_REGION

REGION Network 403: Area A7 =SC00+UC271.GF006 - GF001 POWER CUT UC271 LINE
   "FDBACK_=SC00+UC27.EL001-Q32001/Q32002"(ON := "05_EM_STATE".A7_EMERGENCY_DELAY,   // FDBACK
                           FEEDBACK := "=SC00+UC27.EL001-Q32002 ( =SC00+UC271.GF006 - GF001 BELTS)",
                           QBAD_FIO := NOT "QBAD =SC00+UC27.EL001-Q32001/Q32002",
                           ACK_NEC := true,
                           ACK := "05_EM_STATE".A7_RESET,
                           FDB_TIME := T#300ms,
                           Q => "=SC00+UC27.EL001-Q32001 (=SC00+UC271.GF006 - GF001)");
END_REGION

REGION Network 404: Area A7 =SC00+UC272.RB008 - GF001 POWER CUT UC272 LINE
   "FDBACK_=SC00+UC27.EL001-Q32003/Q32004"(ON := "05_EM_STATE".A7_EMERGENCY_DELAY,   // FDBACK
                           FEEDBACK := "=SC00+UC27.EL001-Q32004 ( =SC00+UC272.RB008 - GF001 BELTS)",
                           QBAD_FIO := NOT "QBAD =SC00+UC27.EL001-Q32003/Q32004",
                           ACK_NEC := true,
                           ACK := "05_EM_STATE".A7_RESET,
                           FDB_TIME := T#300ms,
                           Q => "=SC00+UC27.EL001-Q32003 (=SC00+UC272.RB008 - GF001)");
END_REGION

REGION Network 405: Area A7 =SC00+UC273.GF001 - GF008 POWER CUT UC273 LINE
   "FDBACK_=SC00+UC27.EL001-Q32101/Q32102"(ON := "05_EM_STATE".A7_EMERGENCY_DELAY,   // FDBACK
                           FEEDBACK := "=SC00+UC27.EL001-Q32102 ( =SC00+UC273.GF001 - GF008 BELTS)",
                           QBAD_FIO := NOT "QBAD =SC00+UC27.EL001-Q32101/Q32102",
                           ACK_NEC := true,
                           ACK := "05_EM_STATE".A7_RESET,
                           FDB_TIME := T#300ms,
                           Q => "=SC00+UC27.EL001-Q32101 (=SC00+UC273.GF001 - GF008)");
END_REGION
END_FUNCTION
